Universal Robots URScript: test1.urscript

def test():

movej([0, -1.57079632, 0, -1.57079632, 0, 0],a=0.1,v=0.05)

end
